TYPE "Type_IOParam"
VERSION : 0.1
   STRUCT
      "name" : String["DIM_STRINGNAME"];
      iotype : Int := -1;   // 0 = DI, 1 = AI, 2 = DO, 3 = AO, 4 = RI
      boolval : Array[0.."MAX_IOBOOL"] of Bool;
      intval : Array[0.."MAX_IOINT"] of Int := [9(-1)];
      dintval : Array[0.."MAX_IODINT"] of DInt;
      realvalcfg : Array[0.."MAX_IOREAL"] of Real := [3(0.0), 3(1.0)];
      realval : Array[0.."MAX_IOREAL"] of Real := [3(0.0), 3(1.0)];
      exprintval : Array[0.."MAX_EXPRINT"] of Int := [25(-1)];   // typ + (not, opnd, oper) x 8
      exprrealval : Array[0.."MAX_EXPROPER"] of Real;
   END_STRUCT;

END_TYPE

